// Implicitly generated code : DO NOT EDIT
FUNCTION CheckRangeSigned : DINT
VAR_INPUT
	value, lower, upper: DINT;
END_VAR

// Implicitly generated code : Only an Implementation suggestion
{noflow}
Fault_Count_G(CU:=FALSE) ; 
IF (value < lower) THEN
	CheckRangeSigned := lower;
		Fault_Count_G(CU:=TRUE) ; 
ELSIF(value > upper) THEN
	CheckRangeSigned := upper;
		Fault_Count_G(CU:=TRUE) ; 
ELSE
	CheckRangeSigned := value;
END_IF
{flow}

END_FUNCTION

(* stored: Version 1.1.0.1, ProductVersion 3.1.4024.2
   POU CheckRangeSigned: Id {ad00f06c-c54b-4001-972a-980472a78990}, SpecialFunc CheckRangeSigned *)
